Staubli VAL3: HOME.dtx

InstrItem tcpInstr
  [0]
    string sType
    string sData
Trajectory tTraj
  [0]
    TrajectoryItem tSuper[3]
      [0]
        num distance
        num moveType
        num nTime
        num nStop
        num nTcpAction
        string comment
        bool toStop
        mdesc nom_speed = {tmax=300, rmax=9999, leave=30, reach=30}
        InstrItem iInstr[3]
          [0]
            string sType
            string sData
          [1]
            string sType
            string sData
          [2]
            string sType
            string sData
        num nMoveId
      [1]
        num distance
        num moveType
        num nTime
        num nStop
        num nTcpAction
        string comment = "@JPOINT jZone1"
        bool toStop
        mdesc nom_speed = {tmax=9999, rmax=9999, leave=30, reach=30}
        InstrItem iInstr[3]
          [0]
            string sType
            string sData
          [1]
            string sType
            string sData
          [2]
            string sType
            string sData
        num nMoveId
      [2]
        num distance
        num moveType = 1
        num nTime
        num nStop
        num nTcpAction
        string comment = "@JPOINT jZone1Out"
        bool toStop
        mdesc nom_speed = {vel=450, tmax=1500, rmax=9999, leave=30, reach=30}
        InstrItem iInstr[3]
          [0]
            string sType
            string sData
          [1]
            string sType
            string sData
          [2]
            string sType
            string sData
        num nMoveId
    string sID = "HOME Zone1"
    num nId
public bool bMoveType[3]
  [0] = true
  [1] = true
public bool bStepping
bool bToSave
frame fFrame = {fatherId=world[0]}
frame fSetFrame = {x=-364.286321, y=-1043.316491, z=11.196424, rx=-6.99985, ry=11.31473, rz=18.24134, fatherId=world[0]}
mdesc nom_speed = {accel=25, vel=25, decel=25, blend=off}
num nCoeff = 1
num nDistance = 357.24033
num nHome
num nIndex
num nJoint
num nKey
num nSelected
num nView
num nZeta
pointRx pBestFit[3]
  [0] = {fatherId=world[0]}
  [1] = {fatherId=world[0]}
  [2] = {fatherId=world[0]}
pointRx pCheck = {fatherId=world[0]}
pointRx pNull = {fatherId=world[0]}
pointRx pPointTo = {fatherId=world[0]}
pointRx pPoints[3]
  [0] = {x=-364.286321, y=-1043.316491, z=11.196424, rx=84.453459, ry=18.310573, rz=168.800057, shoulder=lefty, elbow=epositive, wrist=wnegative, fatherId=world[0]}
  [1] = {x=-169.661081, y=-983.133224, z=-35.427424, rx=84.45454, ry=18.311675, rz=168.800636, shoulder=lefty, elbow=epositive, wrist=wnegative, fatherId=world[0]}
  [2] = {x=-263.249747, y=-701.832631, z=-51.099539, rx=84.453256, ry=18.310748, rz=168.801333, shoulder=lefty, elbow=epositive, wrist=wnegative, fatherId=world[0]}
string sInstruction
string sInstruction2
public string sItems[7]
  [0] = "cube_Salle_Bl"
  [1] = "cube_evac_rebut"
  [2] = "cube_moule"
  [3] = "cube_prelev"
  [4] = "home"
string sJoint = "Pt_Pass_Centre"
string sJointCycle = "Pt_Pass_Centre"
string sList
string sMessage
string sPoint = "Centre_Moule"
string sPointCycle = "Centre_Moule"
string sTrajType = "HOME"
trsf tAppro
trsf tPointTo
mdesc mMdesc = {accel=10, vel=10, decel=10, blend=off}
TrajHome jEditPoint
  [0]
    num nIndexTool
    TrajJointItem tData
      [0]
        jointRx jJoint
        TrajectoryItem tSuper
          [0]
            num distance
            num moveType
            num nTime
            num nStop
            num nTcpAction
            string comment
            bool toStop
            mdesc nom_speed = {accel=50, vel=50, decel=50, tmax=300, rmax=9999, leave=30, reach=30}
            InstrItem iInstr[3]
              [0]
                string sType
                string sData
              [1]
                string sType
                string sData
              [2]
                string sType
                string sData
            num nMoveId
    string sID
    num nZoneType
    num nZoneMove
    pointRx pO
    pointRx pX
    pointRx pY
    num nDimension
    pointRx pPointMove
    frame fFrame
    string sProgram
    num nIndexFrame
string sTrajCycle
